              if(rq_write_lgn[index] == -1 and rq_read_lgn[index] != -1):
                  rq_write_lgn[index] = rq_read_lgn[index]
                  rq_write_lgn_previous[index] = rq_read_lgn[index]
              elif(rq_write_lgn_previous[index] == -1 and rq_read_lgn[index] != -1):
                  rq_write_lgn_previous[index] = rq_read_lgn[index]
              end

              if(rq_write_msc[index] == -1 and rq_read_msc[index] != -1):
                  rq_write_msc[index] = rq_read_msc[index]
                  rq_write_msc_previous[index] = rq_read_msc[index]
              elif(rq_write_msc_previous[index] == -1 and rq_read_msc[index] != -1):
                  rq_write_msc_previous[index] = rq_read_msc[index]
              end

              if(rq_write_mod[index] == -1 and rq_read_mod[index] != -1):
                  rq_write_mod[index] = rq_read_mod[index]
                  rq_write_mod_previous[index] = rq_read_mod[index]
              elif(rq_write_mod_previous[index] == -1 and rq_read_mod[index] != -1):
                  rq_write_mod_previous[index] = rq_read_mod[index]
              end

          end
          index = index + 1
      end
  end

  def rq_comm_set_var(var, value=0, gripper_socket="1"):
      socket_set_var(var, value, gripper_socket)
      return socket_read_byte_list(3, gripper_socket)
  end

  def rq_comm_set_pos_spe_for(pos=0, speed=0, force=0, gripper_socket="1"):
      socket_send_string("SET POS", gripper_socket)
      socket_send_byte(32, gripper_socket)
      socket_send_string(pos, gripper_socket)
      socket_send_byte(32, gripper_socket)
      socket_send_string("SPE", gripper_socket)
      socket_send_byte(32, gripper_socket)
      socket_send_string(speed, gripper_socket)
      socket_send_byte(32, gripper_socket)
      socket_send_string("FOR", gripper_socket)
      socket_send_byte(32, gripper_socket)
      socket_send_string(force, gripper_socket)
      socket_send_byte(10, gripper_socket)
      return socket_read_byte_list(3, gripper_socket)
  end

  def rq_comm_read_variables():
      index = 0

      while(index <= 3):
          socket = rq_index_to_socket(index)

          if(gripper_connected[index]):

              if(rq_read_act_req[index]):
                  rq_read_act[index] = socket_get_var("ACT", socket)
                  rq_read_act_req[index] = False
              end

              if(rq_read_gto_req[index]):
                  rq_read_gto[index] = socket_get_var("GTO", socket)
                  rq_read_gto_req[index] = False
              end

              if(rq_read_pre_req[index]):
                  rq_read_pre[index] = socket_get_var("PRE", socket)
                  rq_read_pre_req[index] = False
              end

              if(rq_read_pos_req[index]):
                  rq_read_pos[index] = socket_get_var("POS", socket)
                  rq_read_pos_req[index] = False
              end

              if(rq_read_spe_req[index]):
                  rq_read_spe[index] = socket_get_var("SPE", socket)
                  rq_read_spe_req[index] = False
              end

              if(rq_read_for_req[index]):
                  rq_read_for[index] = socket_get_var("FOR", socket)
                  rq_read_for_req[index] = False
              end

              if(rq_read_obj_req[index]):
                  rq_read_obj[index] = socket_get_var("OBJ", socket)
                  rq_read_obj_req[index] = False
              end

              if(rq_read_sta_req[index]):
                  rq_read_sta[index] = socket_get_var("STA", socket)
                  rq_read_sta_req[index] = False
              end

              if(rq_read_mod_req[index]):
                  rq_read_mod[index] = socket_get_var("MOD", socket)
                  rq_read_mod_req[index] = False
              end

              if(rq_read_flt_req[index]):
                  rq_read_flt[index] = socket_get_var("FLT",socket)
                  rq_read_flt_req[index] = False
              end

              if(rq_read_lbp_req[index]):
                  rq_read_lbp[index] = socket_get_var("LBP", socket)
                  rq_read_lbp_req[index] = False
              end

              if(rq_read_lrd_req[index]):
                  rq_read_lrd[index] = socket_get_var("LRD", socket)
                  rq_read_lrd_req[index] = False
              end

              if(rq_read_lbl_req[index]):
                  rq_read_lbl[index] = socket_get_var("LBL",socket)
                  rq_read_lbl_req[index] = False
              end

              if(rq_read_lgn_req[index]):
                  rq_read_lgn[index] = socket_get_var("LGN", socket)
                  rq_read_lgn_req[index] = False
              end

              if(rq_read_msc_req[index]):
                  rq_read_msc[index] = socket_get_var("MSC", socket)
                  rq_read_msc_req[index] = False
              end

              if(rq_read_cou_req[index]):
                  rq_read_cou[index] = socket_get_var("COU", socket)
                  rq_read_cou_req[index] = False
              end

              if(rq_read_ncy_req[index]):
                  rq_read_ncy[index] = socket_get_var("NCY", socket)
                  rq_read_ncy_req[index] = False
              end

              if(rq_read_dst_req[index]):
                  rq_read_dst[index] = socket_get_var("DST", socket)
                  rq_read_dst_req[index] = False
              end

              if(rq_read_pco_req[index]):
                  rq_read_pco[index] = socket_get_var("PCO", socket)
                  rq_read_pco_req[index] = False
              end
          end
          index = index + 1
      end
  end

  def rq_comm_read_constants():

      if(gripper_connected[0]):
          while(rq_read_snu_1 == rq_string_initial_value):
              socket_send_string("GET SNU", "1")
              rq_read_snu_1 = socket_read_string("1")
          end

          while(rq_read_fwv_1 == rq_string_initial_value):
              socket_send_string("GET FWV", "1")
              rq_read_fwv_1 = socket_read_string("1")
          end

          while(rq_read_ver_1 == rq_string_initial_value):
              socket_send_string("GET VER", "1")
              rq_read_ver_1 = socket_read_string("1")
          end
      end

      if(gripper_connected[1]):
          while(rq_read_snu_2 == rq_string_initial_value):
              socket_send_string("GET SNU", "2")
              rq_read_snu_2 = socket_read_string("2")
          end

          while(rq_read_fwv_2 == rq_string_initial_value):
              socket_send_string("GET FWV", "2")
              rq_read_fwv_2 = socket_read_string("2")
          end

          while(rq_read_ver_2 == rq_string_initial_value):
              socket_send_string("GET VER", "2")
              rq_read_ver_2 = socket_read_string("2")
          end
      end

      if(gripper_connected[2]):
          while(rq_read_snu_3 == rq_string_initial_value):
              socket_send_string("GET SNU", "3")
              rq_read_snu_3 = socket_read_string("3")
          end

          while(rq_read_fwv_3 == rq_string_initial_value):
              socket_send_string("GET FWV", "3")
              rq_read_fwv_3 = socket_read_string("3")
          end

          while(rq_read_ver_3 == rq_string_initial_value):
              socket_send_string("GET VER", "3")
              rq_read_ver_3 = socket_read_string("3")
          end
      end

      if(gripper_connected[3]):
          while(rq_read_snu_4 == rq_string_initial_value):
              socket_send_string("GET SNU", "4")
              rq_read_snu_4 = socket_read_string("4")
          end

          while(rq_read_fwv_4 == rq_string_initial_value):
              socket_send_string("GET FWV", "4")
              rq_read_fwv_4 = socket_read_string("4")
          end

          while(rq_read_ver_4 == rq_string_initial_value):
              socket_send_string("GET VER", "4")
              rq_read_ver_4 = socket_read_string("4")
          end
      end
  end

  def rq_comm_write_variables():
      index = 0

      while(index <= 3):
          socket = rq_index_to_socket(index)

          if(gripper_connected[index]):

              if(rq_write_act_request[index]):
                  if(is_ack(rq_comm_set_var("ACT", rq_write_act[index], socket))):
                      rq_write_act_previous[index] = rq_write_act[index]
                      rq_write_act_request[index] = False
                  end
              end

              if(rq_write_gto_request[index]):
                  if(is_ack(rq_comm_set_var("GTO", rq_write_gto[index], socket))):
                      rq_write_gto_previous[index] = rq_write_gto[index]
                      rq_write_gto_request[index] = False
                  end
              end

              if(rq_write_atr_request[index]):
                  if(is_ack(rq_comm_set_var("ATR", rq_write_atr[index], socket))):
                      rq_write_atr_previous[index] = rq_write_atr[index]
                      rq_write_atr_request[index] = False
                  end
              end

              if(rq_write_ard_request[index]):
                  if(is_ack(rq_comm_set_var("ARD", rq_write_ard[index], socket))):
                      rq_write_ard_previous[index] = rq_write_ard[index]
                      rq_write_ard_request[index] = False
                  end
              end

              if(rq_write_pos_request[index]):
                  if(is_ack(rq_comm_set_pos_spe_for(rq_write_pos[index], rq_write_spe[index], rq_write_for[index], socket))):
                      rq_write_pos_previous[index] = rq_write_pos[index]
                      rq_write_spe_previous[index] = rq_write_spe[index]
                      rq_write_for_previous[index] = rq_write_for[index]
                      rq_write_pos_request[index] = False
                  end
              end

              if(rq_write_lbp_request[index]):
                  if(is_ack(rq_comm_set_var("LBP", rq_write_lbp[index], socket))):
                      rq_write_lbp_previous[index] = rq_write_lbp[index]
                      rq_write_lbp_request[index] = False
                  end
              end

              if(rq_write_lrd_request[index]):
                  if(is_ack(rq_comm_set_var("LRD", rq_write_lrd[index], socket))):
                      rq_write_lrd_previous[index] = rq_write_lrd[index]
                      rq_write_lrd_request[index] = False
                  end
              end

              if(rq_write_lbl_request[index]):
                  if(is_ack(rq_comm_set_var("LBL", rq_write_lbl[index], socket))):
                      rq_write_lbl_previous[index] = rq_write_lbl[index]
                      rq_write_lbl_request[index] = False
                  end
              end

              if(rq_write_lgn_request[index]):
                  if(is_ack(rq_comm_set_var("LGN", rq_write_lgn[index], socket))):
                      rq_write_lgn_previous[index] = rq_write_lgn[index]
                      rq_write_lgn_request[index] = False
                  end
              end

              if(rq_write_msc_request[index]):
                  if(is_ack(rq_comm_set_var("MSC", rq_write_msc[index], socket))):
                      rq_write_msc_previous[index] = rq_write_msc[index]
                      rq_write_msc_request[index] = False
                  end
              end

              if(rq_write_mod_request[index]):
                  if(is_ack(rq_comm_set_var("MOD", rq_write_mod[index], socket))):
                      rq_write_mod_previous[index] = rq_write_mod[index]
                      rq_write_mod_request[index] = False
                  end
              end
          end
          index = index + 1
      end
  end

  def rq_activate(gripper_socket="1"):
      if (not rq_is_gripper_activated(gripper_socket)):
          rq_reset(gripper_socket)

          while(not rq_get_var("ACT", 1, gripper_socket) == 0 or not rq_get_var("STA", 1, gripper_socket) == 0):
              rq_reset(gripper_socket)
              sync()
          end

          rq_set_var("ACT",1, gripper_socket)
      end
  end

  def rq_activate_and_wait(gripper_socket="1"):
      if (not rq_is_gripper_activated(gripper_socket)):
          rq_activate(gripper_socket)
          sleep(1.0)

          while(not rq_get_var("ACT", 1, gripper_socket) == 1 or not rq_get_var("STA", 1, gripper_socket) == 3):
              sleep(0.1)
          end

          sleep(0.5)
      end
  end

  def rq_activate_all_grippers(reset=False):
      if(gripper_connected[0]):
          rq_reset_and_activate("1", reset)
      end

      if(gripper_connected[1]):
          rq_reset_and_activate("2", reset)
      end

      if(gripper_connected[2]):
          rq_reset_and_activate("3", reset)
      end

      if(gripper_connected[3]):
          rq_reset_and_activate("4", reset)
      end
  end

  def rq_reset_and_activate(gripper_socket="1", reset=False):
      if(reset):
          rq_reset(gripper_socket)
          rq_activate_and_wait(gripper_socket)
      elif(not rq_is_gripper_activated(gripper_socket)):
          rq_activate_and_wait(gripper_socket)
      end
  end

  def rq_reset(gripper_socket="1"):
      rq_set_var("ACT", 0, gripper_socket)
      rq_set_var("ATR", 0, gripper_socket)

      while(not rq_get_var("ACT", 1, gripper_socket) == 0 or not rq_get_var("STA", 1, gripper_socket) == 0):
          rq_set_var("ACT", 0, gripper_socket)
          rq_set_var("ATR", 0, gripper_socket)
          sync()
      end

      sleep(0.5)
  end

  def rq_auto_release_open_and_wait(gripper_socket="1"):
      rq_set_var("ATR",0, gripper_socket)
      rq_set_var("ARD",0, gripper_socket)
      rq_set_var("ACT",1, gripper_socket)
      sleep(0.1)
      rq_set_var("ATR",1, gripper_socket)

      rq_wait_autorelease_completed(gripper_socket)
  end

  def rq_auto_release_close_and_wait(gripper_socket="1"):
      rq_set_var("ATR",0, gripper_socket)
      rq_set_var("ARD",1, gripper_socket)
      rq_set_var("ACT",1, gripper_socket)
      sleep(0.1)
      rq_set_var("ATR",1, gripper_socket)

      rq_wait_autorelease_completed(gripper_socket)
  end

  def rq_wait_autorelease_completed(gripper_socket="1"):
      remainingRetries = 20
      gFLT = rq_get_var("FLT", 2, gripper_socket)

      while(not is_FLT_autorelease_in_progress(gFLT) and remainingRetries > 0):
          remainingRetries = remainingRetries - 1
          gFLT = rq_get_var("FLT", 2, gripper_socket)
          sleep(0.1)
      end

      remainingRetries = 100
      gFLT = rq_get_var("FLT", 2, gripper_socket)

      while(not is_FLT_autorelease_completed(gFLT) and remainingRetries > 0):
          remainingRetries = remainingRetries - 1
          gFLT = rq_get_var("FLT", 2, gripper_socket)
          sleep(0.1)
      end
  end

  def rq_set_force(force, gripper_socket="1"):
      force = floor(scale(force, [0, 255], [0.0, 255.0]))
      rq_set_var("FOR", force, gripper_socket)
  end

  def rq_set_speed(speed, gripper_socket="1"):
      speed = floor(scale(speed, [0, 255], [0.0, 255.0]))
      rq_set_var("SPE", speed, gripper_socket)
  end

  def rq_open(gripper_socket="1"):
      rq_move(0, gripper_socket)
  end

  def rq_close(gripper_socket="1"):
      rq_move(255, gripper_socket)
  end

  def rq_open_and_wait(gripper_socket="1"):
      rq_move_and_wait(0, gripper_socket)
  end

  def rq_close_and_wait(gripper_socket="1"):
      rq_move_and_wait(255, gripper_socket)
  end

  def rq_move(pos, gripper_socket="1"):
      rq_set_pos(pos, gripper_socket)
      rq_go_to(gripper_socket)
  end

  def rq_move_and_wait(pos, gripper_socket="1"):
      rq_move(pos, gripper_socket)

      while (not rq_is_motion_complete(gripper_socket)):
          # wait for motion completed
          sync()
      end
  end

  def rq_wait_for_pos_request(pos, gripper_socket="1"):
      gPRE = rq_get_var("PRE", 3, gripper_socket)

      while (gPRE != pos):
          rq_set_var("POS", pos, gripper_socket)
          sync()
          gPRE = rq_get_var("PRE", 3, gripper_socket)
      end
  end

  def rq_wait_pos_spe_for_request(pos, speed, force, gripper_socket="1"):
      gPRE = rq_get_var("PRE", 3, gripper_socket)

      while (gPRE != pos):
          rq_set_pos_spe_for_var(pos, speed, force, gripper_socket)
          sync()
          gPRE = rq_get_var("PRE", 3, gripper_socket)
      end
  end

  def rq_wait_for_pos(pos, gripper_socket="1"):
      rq_wait_for_pos_request(pos, gripper_socket)

      # Wait for the gripper motion to complete
      while (not rq_is_motion_complete(gripper_socket)):
          # wait for motion completed
          sync()
          rq_set_var("GTO", 1, gripper_socket)
      end
  end

  def rq_wait(gripper_socket="1"):
      # Wait for the gripper motion to complete
      while (not rq_is_motion_complete(gripper_socket)):
          sync()
          # The following patch is for Robotiq's Camera issue when communication is lost, but not the activation
          # the communication driver reset the GTO bit
          rq_set_var("GTO", 1, gripper_socket)
      end
  end

  def rq_wait_for_object_detected(gripper_socket="1"):
      # Wait the object detection
      while (not rq_is_object_detected(gripper_socket)):
          sync()
      end
  end

  # set the position
  def rq_set_pos(pos, gripper_socket="1"):
      pos = floor(scale(pos, [0, 255], [0.0, 255.0]))
      rq_set_var("POS", pos, gripper_socket)
      rq_wait_for_pos_request(pos, gripper_socket)
  end

  def rq_set_pos_spd_for(pos, speed, force, gripper_socket="1"):
      pos = floor(scale(pos, [0, 255], [0.0, 255.0]))
      speed = floor(scale(speed, [0, 255], [0.0, 255.0]))
      force = floor(scale(force, [0, 255], [0.0, 255.0]))

      rq_set_pos_spe_for_var(pos, speed, force, gripper_socket)
  end

  def rq_set_gripper_max_current_mA(current_mA, gripper_socket="1"):
      current = floor(current_mA / 10)

      rq_set_var("MSC", current, gripper_socket)
      current_read = rq_get_var("MSC", 1, gripper_socket)

      while(current_read != current):
          rq_set_var("MSC", current, gripper_socket)
          current_read = rq_get_var("MSC", 1, gripper_socket)
      end
  end

  def rq_set_gripper_mode(mode, gripper_socket="1"):
      rq_set_var("MOD", mode, gripper_socket)
  end

  def rq_set_gripper_max_cur(current_mA, gripper_socket="1"):
      rq_set_gripper_max_current_mA(current_mA, gripper_socket)
  end

  def rq_get_gripper_max_current_mA(gripper_socket="1"):
      current = rq_get_var("MSC", 1, gripper_socket)

      if(current == -1):
          current_mA = current
      else:
          current_mA = current * 10
      end

      return current_mA
  end

  def rq_get_gripper_max_cur(gripper_socket="1"):
      return rq_get_gripper_max_current_mA(gripper_socket)
  end

  def rq_set_max_current_for_all_grippers():
      current_mA = rq_get_max_current_mA()

      if(gripper_connected[0]):
          rq_set_gripper_max_current_mA(current_mA, "1")
      end

      if(gripper_connected[1]):
          rq_set_gripper_max_current_mA(current_mA, "2")
      end

      if(gripper_connected[2]):
          rq_set_gripper_max_current_mA(current_mA, "3")
      end

      if(gripper_connected[3]):
          rq_set_gripper_max_current_mA(current_mA, "4")
      end
  end

  def rq_get_max_current_mA():
      max_current_mA = 0

      if(rq_current_limit_enabled):
          nb_connected_grippers = rq_get_nb_connected_grippers()

          if(nb_connected_grippers == 1):
              max_current_mA = 600
          elif(nb_connected_grippers > 1):
              max_current_mA = 450
          end
      else:

      end

      return max_current_mA
  end

  def rq_get_nb_connected_grippers():
      nb_connected_grippers = 0

      if(gripper_connected[0]):
          nb_connected_grippers = nb_connected_grippers + 1
      end

      if(gripper_connected[1]):
          nb_connected_grippers = nb_connected_grippers + 1
      end

      if(gripper_connected[2]):
          nb_connected_grippers = nb_connected_grippers + 1
      end

      if(gripper_connected[3]):
          nb_connected_grippers = nb_connected_grippers + 1
      end

      return nb_connected_grippers
  end

  def rq_list_of_bytes_to_value(list_of_bytes):
      value = -1

      # response list length
      if (list_of_bytes[0] == 1):
          value = list_of_bytes[1] - 48
      elif (list_of_bytes[0] == 2):
          value = (list_of_bytes[1] - 48) * 10 + (list_of_bytes[2] - 48)
      elif (list_of_bytes[0] == 3):
          value = (list_of_bytes[1] - 48) * 100 + (list_of_bytes[2] - 48) * 10 + (list_of_bytes[3] - 48)
      end

      return value
  end

  def rq_is_motion_complete(gripper_socket="1"):
      gOBJ = rq_get_var("OBJ", 1, gripper_socket)
      sync()
      return is_OBJ_gripper_at_position(gOBJ) or is_OBJ_object_detected(gOBJ)
  end

  def rq_is_gripper_activated(gripper_socket="1"):
      gSTA = rq_get_var("STA", 1, gripper_socket)
      sync()
      return is_STA_gripper_activated(gSTA)
  end

  def rq_is_object_detected(gripper_socket="1"):
      gOBJ = rq_get_var("OBJ", 1, gripper_socket)
      sync()
      return is_OBJ_object_detected(gOBJ)
  end

  def rq_current_pos(gripper_socket="1"):
      gPOS = rq_get_var("POS", 1, gripper_socket)
      sync()
      return gPOS
  end

  def rq_motor_current(gripper_socket="1"):
      rq_current = rq_get_var("COU", 1, gripper_socket)
      sync()
      return rq_current * 10
  end

  def rq_print_connected_grippers():
      if(gripper_connected[0]):
          textmsg("Gripper 1 : ", "connected and socket open.")
      end

      if (gripper_connected[1]):
          textmsg("Gripper 2 : ", "connected and socket open.")
      end

      if (gripper_connected[2]):
          textmsg("Gripper 3 : ", "connected and socket open.")
      end

      if (gripper_connected[3]):
          textmsg("Gripper 4 : ", "connected and socket open.")
      end
  end

  def rq_print_gripper_fault_code(gripper_socket="1"):
      gFLT = rq_get_var("FLT", 2, gripper_socket)

      if(is_FLT_no_fault(gFLT)):
          textmsg("Gripper Fault : ", "No Fault (0x00)")
      elif (is_FLT_action_delayed(gFLT)):
          textmsg("Gripper Fault : ", "Priority Fault: Action delayed, initialization must be completed prior to action (0x05)")
      elif (is_FLT_not_activated(gFLT)):
          textmsg("Gripper Fault : ", "Priority Fault: The activation must be set prior to action (0x07)")
      elif (is_FLT_autorelease_in_progress(gFLT)):
          textmsg("Gripper Fault : ", "Minor Fault: Automatic release in progress (0x0B)")
      elif (is_FLT_overcurrent(gFLT)):
          textmsg("Gripper Fault : ", "Minor Fault: Overcurrent protection triggered (0x0E)")
      elif (is_FLT_autorelease_completed(gFLT)):
          textmsg("Gripper Fault : ", "Major Fault: Automatic release completed (0x0F)")
      else:
          textmsg("Gripper Fault : ", "Unknown Fault")
      end
  end

  def rq_print_gripper_num_cycles(gripper_socket="1"):
      num_cycles = rq_get_var("NCY", 1, gripper_socket)

      if(num_cycles == -1):
          textmsg("Gripper Cycle Number : ", "Number of cycles is unreachable.")
      else:
          textmsg("Gripper Cycle Number : ", num_cycles)
      end
  end

  def rq_print_gripper_driver_state(gripper_socket="1"):
      driver_state = rq_get_var("DST", 1, gripper_socket)

      if(driver_state == 0):
          textmsg("Gripper Driver State : ", "RQ_STATE_INIT")
      elif(driver_state == 1):
          textmsg("Gripper Driver State : ", "RQ_STATE_LISTEN")
      elif(driver_state == 2):
          textmsg("Gripper Driver State : ", "RQ_STATE_READ_INFO")
      elif(driver_state == 3):
          textmsg("Gripper Driver State : ", "RQ_STATE_ACTIVATION")
      else:
          textmsg("Gripper Driver State : ", "RQ_STATE_RUN")
      end
  end

  def rq_print_gripper_serial_number(gripper_socket="1"):
      serial_number = rq_get_var_string("SNU", 1, gripper_socket)
      textmsg("Gripper Serial Number : ", serial_number)
  end

  def rq_print_gripper_firmware_version(gripper_socket="1"):
      firmware_version = rq_get_var_string("FWV", 1, gripper_socket)
      textmsg("Gripper Firmware Version : ", firmware_version)
  end

  def rq_print_gripper_driver_version(gripper_socket="1"):
      driver_version = rq_get_var_string("VER", 1, gripper_socket)
      textmsg("Gripper Driver Version : ", driver_version)
  end

  def rq_print_gripper_connection_state(gripper_socket="1"):
      connection_state = rq_get_var("PCO", 1, gripper_socket)

      if (connection_state == 0):
          textmsg("Gripper Connection State : ", "No connection problem detected")
      else:
          textmsg("Gripper Connection State : ", "Connection problem detected")
      end
  end

  # Returns True if list_of_bytes is [3, 'a', 'c', 'k']
  def is_ack(list_of_bytes):

      # list length is not 3
      if (list_of_bytes[0] != 3):
          return False
      end

      # first byte not is 'a'?
      if (list_of_bytes[1] != 97):
          return False
      end

      # first byte not is 'c'?
      if (list_of_bytes[2] != 99):
          return False
      end

      # first byte not is 'k'?
      if (list_of_bytes[3] != 107):
          return False
      end

      return True
  end

  # Returns True if list_of_bytes is not [3, 'a', 'c', 'k']
  def is_not_ack(list_of_bytes):
      if (is_ack(list_of_bytes)):
          return False
      else:
          return True
      end
  end

  def is_STA_gripper_activated (gSTA):
      if (gSTA == 3):
          return True
      end

      return False
  end

  def is_OBJ_object_detected (gOBJ):
      if (gOBJ == 1 or gOBJ == 2):
          return True
      end

      return False
  end

  def is_OBJ_gripper_at_position (gOBJ):
      if (gOBJ == 3):
          return True
      end

      return False
  end

  def is_not_OBJ_gripper_at_position (gOBJ):
      if (is_OBJ_gripper_at_position(gOBJ)):
          return False
      else:
          return True
      end
  end

  #### GTO Section ####
  def rq_stop(gripper_socket="1"):
      rq_set_var("GTO", 0, gripper_socket)
  end

  def rq_set_GTO_and_wait(value, gripper_socket="1"):
      rq_set_var("GTO" ,value, gripper_socket)
      while(not is_GTO(value, rq_get_var("GTO", 1, gripper_socket))):
        sync()
      end
  end

  def rq_go_to(gripper_socket="1"):
      rq_set_var("GTO", 1, gripper_socket)
  end


  def is_GTO(goto_value, rGTO):
      return rGTO == goto_value
  end
  #### GTO Section ####

  def is_FLT_no_fault(gFLT):
      return gFLT == 0
  end

  def is_FLT_warning(gFLT):
      return gFLT >= 1 and gFLT <= 7
  end

  def is_FLT_faulted(gFLT):
      return gFLT >= 8
  end

  def is_FLT_action_delayed(gFLT):
      return gFLT == 5
  end

  def is_FLT_not_activated(gFLT):
      return gFLT == 7
  end

  def is_FLT_autorelease_in_progress(gFLT):
      return gFLT == 11
  end

  def is_FLT_overcurrent(gFLT):
      return gFLT == 14
  end

  def is_FLT_autorelease_completed(gFLT):
      return gFLT == 15
  end

  def rq_set_var(var_name, var_value, gripper_socket="1"):
      index = rq_socket_to_index(gripper_socket)

      enter_critical

      if (var_name == "ACT"):
          rq_write_act[index] = var_value
          rq_write_act_request[index] = True
      elif (var_name == "GTO"):
          rq_write_gto[index] = var_value
          rq_write_gto_request[index] = True
      elif (var_name == "ATR"):
          rq_write_atr[index] = var_value
          rq_write_atr_request[index] = True
      elif (var_name == "ARD"):
          rq_write_ard[index] = var_value
          rq_write_ard_request[index] = True
      elif (var_name == "FOR"):
          rq_write_for[index] = var_value
          rq_write_pos_request[index] = True
      elif (var_name == "SPE"):
          rq_write_spe[index] = var_value
          rq_write_pos_request[index] = True
      elif (var_name == "POS"):
          rq_write_pos[index] = var_value
          rq_write_pos_request[index] = True
      elif (var_name == "LBP"):
          rq_write_lbp[index] = var_value
          rq_write_lbp_request[index] = True
      elif (var_name == "LRD"):
          rq_write_lrd[index] = var_value
          rq_write_lrd_request[index] = True
      elif (var_name == "LBL"):
          rq_write_lbl[index] = var_value
          rq_write_lbl_request[index] = True
      elif (var_name == "LGN"):
          rq_write_lgn[index] = var_value
          rq_write_lgn_request[index] = True
      elif (var_name == "MSC"):
          rq_write_msc[index] = var_value
          rq_write_msc_request[index] = True
      elif (var_name == "MOD"):
          rq_write_mod[index] = var_value
          rq_write_mod_request[index] = True
      end

      exit_critical

      if (var_name == "ACT"):
          while(rq_write_act_request[index]):
              sync()
          end
      elif (var_name == "GTO"):
          while(rq_write_gto_request[index]):
              sync()
          end
      elif (var_name == "ATR"):
          while(rq_write_atr_request[index]):
              sync()
          end
      elif (var_name == "ARD"):
          while(rq_write_ard_request[index]):
              sync()
          end
      elif (var_name == "FOR"):
          while(rq_write_pos_request[index]):
              sync()
          end
      elif (var_name == "SPE"):
          while(rq_write_pos_request[index]):
              sync()
          end
      elif (var_name == "POS"):
          while(rq_write_pos_request[index]):
              sync()
          end
      elif (var_name == "LBP"):
          while(rq_write_lbp_request[index]):
              sync()
          end
      elif (var_name == "LRD"):
          while(rq_write_lrd_request[index]):
              sync()
          end
      elif (var_name == "LBL"):
          while(rq_write_lbl_request[index]):
              sync()
          end
      elif (var_name == "LGN"):
          while(rq_write_lgn_request[index]):
              sync()
          end
      elif (var_name == "MSC"):
          while(rq_write_msc_request[index]):
              sync()
          end
      elif (var_name == "MOD"):
          while(rq_write_mod_request[index]):
              sync()
          end
      end
  end

  def rq_set_pos_spe_for_var(pos, speed, force, gripper_socket="1"):
      index = rq_socket_to_index(gripper_socket)

      enter_critical

      rq_write_for[index] = force
      rq_write_spe[index] = speed
      rq_write_pos[index] = pos
      rq_write_pos_request[index] = True

      exit_critical
  end

  def rq_get_var(var_name, nbr_bytes, gripper_socket="1"):
      index = rq_socket_to_index(gripper_socket)
      var_value = -1

      if (var_name == "ACT"):
          enter_critical
          rq_read_act_req[index] = True
          exit_critical
          while(rq_read_act_req[index]):
              sync()
          end
          var_value = rq_read_act[index]

      elif (var_name == "GTO"):
          enter_critical
          rq_read_gto_req[index] = True
          exit_critical
          while(rq_read_gto_req[index]):
              sync()
          end
          var_value = rq_read_gto[index]

      elif (var_name == "FOR"):
          enter_critical
          rq_read_for_req[index] = True
          exit_critical
          while(rq_read_for_req[index]):
              sync()
          end
          var_value = rq_read_for[index]

      elif (var_name == "SPE"):
          enter_critical
          rq_read_spe_req[index] = True
          exit_critical
          while(rq_read_spe_req[index]):
              sync()
          end
          var_value = rq_read_spe[index]

      elif (var_name == "OBJ"):
          enter_critical
          rq_read_obj_req[index] = True
          exit_critical
          while(rq_read_obj_req[index]):
              sync()
          end
          var_value = rq_read_obj[index]

      elif (var_name == "STA"):
          enter_critical
          rq_read_sta_req[index] = True
          exit_critical
          while(rq_read_sta_req[index]):
              sync()
          end
          var_value = rq_read_sta[index]

      elif (var_name == "FLT"):
          enter_critical
          rq_read_flt_req[index] = True
          exit_critical
          while(rq_read_flt_req[index]):
              sync()
          end
          var_value = rq_read_flt[index]

      elif (var_name == "POS"):
          enter_critical
          rq_read_pos_req[index] = True
          exit_critical
          while(rq_read_pos_req[index]):
              sync()
          end
          var_value = rq_read_pos[index]

      elif (var_name == "PRE"):
          enter_critical
          rq_read_pre_req[index] = True
          exit_critical
          while(rq_read_pre_req[index]):
              sync()
          end
          var_value = rq_read_pre[index]

      elif (var_name == "LBP"):
          enter_critical
          rq_read_lbp_req[index] = True
          exit_critical
          while(rq_read_lbp_req[index]):
              sync()
          end
          var_value = rq_read_lbp[index]

      elif (var_name == "LRD"):
          enter_critical
          rq_read_lrd_req[index] = True
          exit_critical
          while(rq_read_lrd_req[index]):
              sync()
          end
          var_value = rq_read_lrd[index]

      elif (var_name == "LBL"):
          enter_critical
          rq_read_lbl_req[index] = True
          exit_critical
          while(rq_read_lbl_req[index]):
              sync()
          end
          var_value = rq_read_lbl[index]

      elif (var_name == "LGN"):
          enter_critical
          rq_read_lgn_req[index] = True
          exit_critical
          while(rq_read_lgn_req[index]):
              sync()
          end
          var_value = rq_read_lgn[index]

      elif (var_name == "MSC"):
          enter_critical
          rq_read_msc_req[index] = True
          exit_critical
          while(rq_read_msc_req[index]):
              sync()
          end
          var_value = rq_read_msc[index]

      elif (var_name == "MOD"):
          enter_critical
          rq_read_mod_req[index] = True
          exit_critical
          while(rq_read_mod_req[index]):
              sync()
          end
          var_value = rq_read_mod[index]

      elif (var_name == "NCY"):
          enter_critical
          rq_read_ncy_req[index] = True
          exit_critical
          while(rq_read_ncy_req[index]):
              sync()
          end
          var_value = rq_read_ncy[index]

      elif (var_name == "PCO"):
          enter_critical
          rq_read_pco_req[index] = True
          exit_critical
          while(rq_read_pco_req[index]):
              sync()
          end
          var_value = rq_read_pco[index]

      elif (var_name == "DST"):
          enter_critical
          rq_read_dst_req[index] = True
          exit_critical
          while(rq_read_dst_req[index]):
              sync()
          end
          var_value = rq_read_dst[index]

      end

      return var_value
  end

  def rq_get_var_string(var_name, nbr_bytes, gripper_socket="1"):
      index = rq_socket_to_index(gripper_socket)
      var_value = ""

      enter_critical

      if (var_name == "SNU"):
          if(gripper_socket == "1"):
              var_value = rq_read_snu_1
          elif(gripper_socket == "2"):
              var_value = rq_read_snu_2
          elif(gripper_socket == "3"):
              var_value = rq_read_snu_3
          elif(gripper_socket == "4"):
              var_value = rq_read_snu_4
          end
      elif (var_name == "FWV"):
          if(gripper_socket == "1"):
              var_value = rq_read_fwv_1
          elif(gripper_socket == "2"):
              var_value = rq_read_fwv_2
          elif(gripper_socket == "3"):
              var_value = rq_read_fwv_3
          elif(gripper_socket == "4"):
              var_value = rq_read_fwv_4
          end
      elif (var_name == "VER"):
          if(gripper_socket == "1"):
              var_value = rq_read_ver_1
          elif(gripper_socket == "2"):
              var_value = rq_read_ver_2
          elif(gripper_socket == "3"):
              var_value = rq_read_ver_3
          elif(gripper_socket == "4"):
              var_value = rq_read_ver_4
          end
      end

      exit_critical

      return var_value
  end

  def rq_is_object_validated(gripper_selected, gripper_socket="1"):
      if(gripper_selected):
          if(rq_is_object_detected(gripper_socket)):
              return True
          else:
              return False
          end
      else:
          return True
      end
  end

  ############################################
  # normalized functions (maps 0-100 to 0-255)
  ############################################
  def rq_set_force_norm(force_norm, gripper_socket="1"):
      force_gripper = norm_to_gripper(force_norm)
      rq_set_force(force_gripper, gripper_socket)
  end

  def rq_set_speed_norm(speed_norm, gripper_socket="1"):
      speed_gripper = norm_to_gripper(speed_norm)
      rq_set_speed(speed_gripper, gripper_socket)
  end

  def rq_move_norm(pos_norm, gripper_socket="1"):
      pos_gripper = norm_to_gripper(pos_norm)
      rq_move(pos_gripper, gripper_socket)
  end

  def rq_move_and_wait_norm(pos_norm, gripper_socket="1"):
      pos_gripper = norm_to_gripper(pos_norm)
      rq_move_and_wait(pos_gripper, gripper_socket)
  end

  def rq_set_pos_norm(pos_norm, gripper_socket="1"):
      pos_gripper = norm_to_gripper(pos_norm)
      rq_set_pos(pos_gripper, gripper_socket)
  end

  def rq_current_pos_norm(gripper_socket="1"):
      pos_gripper = rq_current_pos(gripper_socket)
      pos_norm = gripper_to_norm(pos_gripper)
      return pos_norm
  end

  def gripper_to_norm(value_gripper):
      value_norm = (value_gripper / 255) * 100
      return floor(value_norm)
  end

  def norm_to_gripper(value_norm):
      value_gripper = (value_norm / 100) * 255
      return ceil(value_gripper)
  end

  def rq_get_position():
      return rq_current_pos_norm()
  end

  def rq_gripper_led_on(gripper_socket="1"):
      rq_set_var("LBP",0, gripper_socket)
  end

  def rq_gripper_led_off(gripper_socket="1"):
      rq_set_var("LBP",1, gripper_socket)
      rq_set_var("LRD",0, gripper_socket)
      rq_set_var("LBL",0, gripper_socket)
      rq_set_var("LGN",0, gripper_socket)
  end

  def rq_gripper_led_force_red(gripper_socket="1"):
      rq_set_var("LBP",1, gripper_socket)
      rq_set_var("LRD",1, gripper_socket)
      rq_set_var("LBL",0, gripper_socket)
      rq_set_var("LGN",0, gripper_socket)
  end

  def rq_gripper_led_force_blue(gripper_socket="1"):
      rq_set_var("LBP",1, gripper_socket)
      rq_set_var("LRD",0, gripper_socket)
      rq_set_var("LBL",1, gripper_socket)
      rq_set_var("LGN",0, gripper_socket)
  end

  def rq_gripper_led_force_green(gripper_socket="1"):
      rq_set_var("LBP",1, gripper_socket)
      rq_set_var("LRD",0, gripper_socket)
      rq_set_var("LBL",0, gripper_socket)
      rq_set_var("LGN",1, gripper_socket)
  end

  def rq_gripper_led_force_purple(gripper_socket="1"):
      rq_set_var("LBP",1, gripper_socket)
      rq_set_var("LRD",1, gripper_socket)
      rq_set_var("LBL",1, gripper_socket)
      rq_set_var("LGN",0, gripper_socket)
  end

  ############################################
  # mm/inches functions
  ############################################
  gripper_closed_norm = [100, 100, 100, 100]
  gripper_open_norm = [0, 0, 0, 0]
  gripper_closed_mm = [0, 0, 0, 0]
  gripper_open_mm = [50, 50, 50, 50]

  def rq_current_pos_mm(gripper_socket=1):
      pos_gripper = rq_current_pos(gripper_socket)
      pos_mm = gripper_to_mm(pos_gripper, gripper_socket)
      return round_value_2_dec(pos_mm)
  end

  def rq_current_pos_inches(gripper_socket=1):
      pos_gripper = rq_current_pos(gripper_socket)
      pos_mm = gripper_to_mm(pos_gripper, gripper_socket)
      pos_in = pos_mm / 25.4
      return round_value_2_dec(pos_in)
  end

  def rq_move_mm(pos_mm, gripper_socket=1):
      pos_gripper = mm_to_gripper(pos_mm, gripper_socket)
      rq_move(pos_gripper, gripper_socket)
  end

  def rq_move_and_wait_mm(pos_mm, gripper_socket=1):
      pos_gripper = mm_to_gripper(pos_mm, gripper_socket)
      rq_move_and_wait(pos_gripper, gripper_socket)
  end

  def rq_move_inches(pos_in, gripper_socket=1):
      pos_mm = pos_in * 25.4
      rq_move_mm(pos_mm, gripper_socket)
  end

  def rq_move_and_wait_inches(pos_in, gripper_socket=1):
      pos_mm = pos_in * 25.4
      rq_move_and_wait_mm(pos_mm, gripper_socket)
  end

  def get_closed_norm(gripper_socket):
      return gripper_closed_norm[gripper_socket - 1]
  end

  def get_open_norm(gripper_socket):
      return gripper_open_norm[gripper_socket - 1]
  end

  def get_closed_mm(gripper_socket):
      return gripper_closed_mm[gripper_socket - 1]
  end

  def get_open_mm(gripper_socket):
      return gripper_open_mm[gripper_socket - 1]
  end

  def set_closed_norm(closed_norm, gripper_socket):
      gripper_closed_norm[gripper_socket - 1] = closed_norm
  end

  def set_open_norm(open_norm, gripper_socket):
      gripper_open_norm[gripper_socket - 1] = open_norm
  end

  def set_closed_mm(closed_mm, gripper_socket):
      gripper_closed_mm[gripper_socket - 1] = closed_mm
  end

  def set_open_mm(open_mm, gripper_socket):
      gripper_open_mm[gripper_socket - 1] = open_mm
  end

  def gripper_to_mm(value_gripper, gripper_socket):
      closed_norm = get_closed_norm(gripper_socket)
      open_norm = get_open_norm(gripper_socket)
      closed_mm = get_closed_mm(gripper_socket)
      open_mm = get_open_mm(gripper_socket)

      value_norm = (value_gripper / 255) * 100

      slope = (closed_mm - open_mm) / (closed_norm - open_norm)
      value_mm = slope * (value_norm - closed_norm) + closed_mm

      if (value_mm > open_mm):
          value_mm_limited = open_mm
      elif (value_mm < closed_mm):
          value_mm_limited = closed_mm
      else:
          value_mm_limited = value_mm
      end

      return value_mm_limited
  end

  def mm_to_gripper(value_mm, gripper_socket):
      closed_norm = get_closed_norm(gripper_socket)
      open_norm = get_open_norm(gripper_socket)
      closed_mm = get_closed_mm(gripper_socket)
      open_mm = get_open_mm(gripper_socket)

      slope = (closed_norm - open_norm) / (closed_mm - open_mm)
      value_norm = (value_mm - closed_mm) * slope + closed_norm

      value_gripper = value_norm * 255 / 100

      if (value_gripper > 255):
          value_gripper_limited = 255
      elif (value_gripper < 0):
          value_gripper_limited = 0
      else:
          value_gripper_limited = round_value(value_gripper)
      end

      return value_gripper_limited
  end

  def round_value(value):
      value_mod = value % 1

      if(value_mod < 0.5):
          return floor(value)
      else:
          return ceil(value)
      end
  end

  def round_value_2_dec(value):
      value_x_100 = value * 100
      value_x_100_rounded = round_value(value_x_100)
      return value_x_100_rounded / 100
  end

  def clear_socket_buffer(gripper_socket="1", read_timeout = 0.1):
      rq_comm_clear_socket_buffer_enabled[rq_socket_to_index(gripper_socket)] = True
  end

  def rq_gripper_id_to_ascii(gripper_id):
      if(gripper_id == "1"):
          return 57
      elif(gripper_id == "2"):
          return 50
      elif(gripper_id == "3"):
          return 51
      elif(gripper_id == "4"):
          return 52
      end
  end

  def scale(value, rawRange, scaledRange):
      def computeSlope(inputRange, outputRange):
          outputRangeDelta = outputRange[1] - outputRange[0]
          inputRangeDelta = inputRange[1] - inputRange[0]

          if (inputRangeDelta == 0):
              return 0
          else:
              return outputRangeDelta / inputRangeDelta
          end
      end

      def computeIntercept(slope, inputRange, outputRange):
          return outputRange[0] - (slope * inputRange[0])
      end

      def clipScaledValue(outputScaledValue, outputRange):
          if (outputRange[0] < outputRange[1]):
              return clipWhenLowerLimitIsLessThanHigher(outputScaledValue, outputRange)
          else:
              return clipWhenLowerLimitIsGreaterThanHigherLimit(outputScaledValue, outputRange)
          end
      end

      def clipWhenLowerLimitIsGreaterThanHigherLimit(outputScaledValue, outputRange):
          if (outputScaledValue < outputRange[1]):
              return outputRange[1]
          elif (outputScaledValue > outputRange[0]):
              return outputRange[0]
          else:
              return outputScaledValue
          end
      end

      def clipWhenLowerLimitIsLessThanHigher(outputScaledValue, outputRange):
          if (outputScaledValue < outputRange[0]):
              return outputRange[0]
          elif (outputScaledValue > outputRange[1]):
              return outputRange[1]
          else:
              return outputScaledValue
          end
      end

      slope = computeSlope(rawRange, scaledRange)
      intercept = computeIntercept(slope, rawRange, scaledRange)
      scaledValue = slope * value + intercept
      return clipScaledValue(scaledValue, scaledRange)
  end

  def limit(value, range):
      return scale(value, range, range)
  end


  rq_init_comm_if_connected(9, "1")
  rq_init_comm_if_connected(2, "2")
  rq_init_comm_if_connected(3, "3")
  rq_init_comm_if_connected(4, "4")
  rq_print_connected_grippers()
  rq_gripper_communication_thread = run rq_gripper_communication()
  set_closed_norm(100.0, 1)
  set_open_norm(0.0, 1)
  set_closed_mm(0.0, 1)
  set_open_mm(50.0, 1)
  set_closed_norm(100.0, 2)
  set_open_norm(0.0, 2)
  set_closed_mm(0.0, 2)
  set_open_mm(50.0, 2)
  set_closed_norm(100.0, 3)
  set_open_norm(0.0, 3)
  set_closed_mm(0.0, 3)
  set_open_mm(50.0, 3)
  set_closed_norm(100.0, 4)
  set_open_norm(0.0, 4)
  set_closed_mm(0.0, 4)
  set_open_mm(50.0, 4)
  rq_current_limit_enabled = False
  while(not rq_gripper_communication_thread_started):
      sync()
  end
  # end: URCap Installation Node
  $ 1 "BeforeStart"
  $ 2 "s_open≔socket_open('192.168.0.10',30000)"
  global s_open=socket_open("192.168.0.10",30000)
  $ 3 "MoveJ"
  $ 4 "pick_pos" "breakAfter"
  movej(get_inverse_kin(p[.419428775081, -.156466791448, .391085213928, 2.180490679377, -2.261344124399, .002804421611], qnear=[0.001867666606264251, -1.1152618567100614, -2.0303900877579535, -1.5673182646379207, 1.5616202354452682, 0.045734424142303]), a=1.3962634015954636, v=1.0471975511965976)
  $ 5 "Loop s_open ≟  False "
  while (s_open  ==    False  ):
    $ 6 "s_open≔socket_open('192.168.0.10',30000)"
    global s_open=socket_open("192.168.0.10",30000)
  end
  $ 7 "robot_start≔'robot start'"
  global robot_start="robot start"
  $ 8 "server_start≔'server start'"
  global server_start="server start"
  $ 9 "part_found≔'part found'"
  global part_found="part found"
  $ 10 "part_n_found≔'part not found'"
  global part_n_found="part not found"
  $ 11 "go_ocr≔'go ocr'"
  global go_ocr="go ocr"
  $ 12 "ocr_position≔'ocr position'"
  global ocr_position="ocr position"
  $ 13 "part_placed≔'part placed'"
  global part_placed="part placed"
  $ 14 "go_pick≔'go pick'"
  global go_pick="go pick"
  $ 15 "var_2≔'0'"
  global var_2="0"
  while (True):
    $ 16 "Robot Program"
    $ 17 "toserver≔robot_start"
    global toserver=robot_start
    $ 18 "socket_send_string(toserver)"
    socket_send_string(toserver)
    $ 19 "Wait: 0.01"
    sleep(0.01)
    $ 20 "fromserver≔socket_read_string()"
    global fromserver=socket_read_string()
    $ 21 "Loop fromserver ≠ server_start"
    while (fromserver  !=  server_start):
      $ 22 "fromserver≔socket_read_string()"
      global fromserver=socket_read_string()
      $ 23 "Wait: 0.01"
      sleep(0.01)
    end
    $ 24 "campos_1"
    $ 25 "Loop"
    while (True):
      $ 26 "MoveJ"
      $ 27 "pick_pos" "breakAfter"
      movej(get_inverse_kin(p[.419428775081, -.156466791448, .391085213928, 2.180490679377, -2.261344124399, .002804421611], qnear=[0.001867666606264251, -1.1152618567100614, -2.0303900877579535, -1.5673182646379207, 1.5616202354452682, 0.045734424142303]), a=1.3962634015954636, v=1.0471975511965976, r=0.1)
      # begin: URCap Program Node
      #   Source: Robotiq_Wrist_Camera, 1.10.3.5692, Robotiq Inc.
      #   Type: Cam Locate
      $ 28 "Cam Locate"

      ###########################################
      #######VisionLocate node start########

      f=[0,0.0,0.0,0.0,0.0,0.0,0.0,0]
      object_location=p[0.0,0.0,0.0,0.0,0.0,0.0]
      feature_pose_to_restore_45951 = pp_n_1
      movej([1.1058803796768188, -1.1670668760882776, -1.9255879561053675, -1.3659794966327112, 1.0898480415344238, 1.0605189800262451])
      # Offset in translation only.
      snapshot_position_offset[3] = 0
      snapshot_position_offset[4] = 0
      snapshot_position_offset[5] = 0
      T_camera_in_flange = p[0, 0, 0, 0, 0, 0] # enlever une fois que l'enseignement du modele sera fait en faisant un movetool avec la pose de la camera dans le repere de la flange. Pour l'instant, on suppose que la camera est situee directement sur la flange.
      tool_45951 = get_T_in_base_from_flange(T_camera_in_flange)
      tool_45951 = pose_sub(tool_45951, snapshot_position_offset)
      snapshot_position = p[0.3857, 0.326079, 0.667286, -1.91141, 1.92966, -0.520215]
      textmsg("expected snapshot position : ", snapshot_position)
      diff = pose_sub(tool_45951, snapshot_position)
      textmsg("diff = ", diff)
      is_at_snapshot_position = norm([diff[0], diff[1], diff[2]]) < 0.002
      is_at_snapshot_position = is_at_snapshot_position and (norm([diff[3], diff[4], diff[5]]) < 0.005)
      textmsg("is_at_snapshot_position = ", is_at_snapshot_position)
      is_snapshot_position_offset = norm(snapshot_position_offset) != 0
      is_at_snapshot_position = is_at_snapshot_position or ignore_snapshot_position
      if not(is_at_snapshot_position):
        popup("Robot is not at Snapshot Position. Add Move instruction to Snapshot Position before Camera Locate node.. Error code: [UCC-8]", warning = False, error = True)
        halt
      end
      f_45951 = xmlrpc_server.findmodel("contextName-45951", tool_45951[0], tool_45951[1], tool_45951[2], tool_45951[3], tool_45951[4], tool_45951[5])
      cam_locate_monitor.setFindModelResult("45951", f_45951)
      canSaveImage = True
      logging_service.publish("FIND_MODEL", f_45951)
      cam_locate_monitor.setCurrentObjectIndex("45951", 0)
      # begin: URCap Program Node
      #   Source: Robotiq_Wrist_Camera, 1.10.3.5692, Robotiq Inc.
      #   Type: Cam Locate Loop
      $ 29 "For object(s) found" "noBreak"
      object_teaching_location_45951 = p[0.3972655139194614, 0.39008004971495547, 0.03268649806528501, -3.1393198709274563, 0.034253799767581854, -2.215684751352942E-5]
      feature_teaching_location_45951 = p[0.3972655139194614, 0.39008004971495547, 0.03268649806528501, -3.1394826802205165, 0.0123293219801983, -4.502308288505037E-5]
      while (not cam_locate_monitor.isCaptureNeeded("45951")):
        poseAsArray = cam_locate_monitor.getCurrentObjectPoseAsArray("45951")
        current_object_location_45951 = p[poseAsArray[0], poseAsArray[1], poseAsArray[2], poseAsArray[3], poseAsArray[4], poseAsArray[5]]
        object_location = current_object_location_45951
        f[0] = cam_locate_monitor.getNumberOfObjectsFound("45951")
        f[1] = object_location[0]
        f[2] = object_location[1]
        f[3] = object_location[2]
        f[4] = object_location[3]
        f[5] = object_location[4]
        f[6] = object_location[5]
        f[7] = cam_locate_monitor.getCurrentObjectDetectionScore("45951")
        textmsg("current_object_location = ", current_object_location_45951)
        if (norm(snapshot_position_offset) != 0):
          current_object_location_45951 = pose_add(current_object_location_45951, snapshot_position_offset)
          textmsg("current_object_location after snapshot position offset = ", current_object_location_45951)
        end
        pp_n_1 = pose_trans(current_object_location_45951, pose_trans(pose_inv(object_teaching_location_45951), feature_teaching_location_45951))
        $ 30 "lp_br≔ False " "noBreak"
        global lp_br=  False
        $ 31 "socket_send_string(part_found)" "noBreak"
        socket_send_string(part_found)
        $ 32 "target≔object_location" "noBreak"
        global target=object_location
        $ 33 "target[2] = target[2] + 0.02" "noBreak"
        target[2] = target[2] + 0.02
        $ 34 "MoveL" "noBreak"
        $ 35 "target" "noBreak"
        movel(pose_trans(p[0.0,0.0,0.0,0.0,0.0,0.0], target), a=1.2, v=0.25)
        # begin: URCap Program Node
        #   Source: Robotiq_Copilot, 1.14.5.5896, Robotiq Inc.
        #   Type: Find Surface
        $ 36 "Find Surface" "noBreak"
        rq_ft_sensor_disconnected_check()
        rq_zero_sensor()
        sleep(0.1)
        surface_found = rq_linear_search_urcap("Z-", 10.000, 0.050, 0.500, 0)
        storevar.setvariable("rq_findSurface_41898b69-db16-4f6d-856e-2ea45cbd8eeb_exitPosition", get_actual_tcp_pose())
        $ 37 "'Add Stop conditions from the Find Surface node'" "noBreak"
        # 'Add Stop conditions from the Find Surface node'
        # end: URCap Program Node
        $ 38 "vac_test≔rq_is_vacuum_obj_detected('1')" "noBreak"
        global vac_test=rq_is_vacuum_obj_detected("1")
        # begin: URCap Program Node
        #   Source: Robotiq_Grippers, 1.8.5.6286, Robotiq Inc.
        #   Type: Vacuum
        $ 39 "Vacuum Grip  (1)           " "noBreak"
        if(not rq_is_gripper_connected("1")):
            popup("A vacuum is not connected. ID: 1", "Vacuum Error", False, True, True)
        end

        rq_vacuum_grip_raw(False, 20, 40, 30, "1")

            suction_completed = rq_wait_for_vacuum_object_suction_complete("1")
            if(not suction_completed):
                rq_set_var("GTO", 0, "1")
            end

        # end: URCap Program Node
        $ 40 "vac_test≔rq_is_vacuum_obj_detected('1')" "noBreak"
        global vac_test=rq_is_vacuum_obj_detected("1")
        $ 41 "If vac_test == False " "noBreak"
        if (vac_test ==  False  ):
          # begin: URCap Program Node
          #   Source: Robotiq_Grippers, 1.8.5.6286, Robotiq Inc.
          #   Type: Vacuum
          $ 42 "Vacuum Release  (1)           " "noBreak"
          if(not rq_is_gripper_connected("1")):
              popup("A vacuum is not connected. ID: 1", "Vacuum Error", False, True, True)
          end

          if(vacuumGripCheckThread1Running):
              stopVacuumGripCheckThread(vacuumGripCheckThread1)
              vacuumGripCheckThread1Running = False
          end

          rq_vacuum_release_raw(False, 100, 60, 30, 0.05, True, "1")

          # end: URCap Program Node
          $ 43 "break" "noBreak"
          break
        end
        # begin: URCap Program Node
        #   Source: Robotiq_Copilot, 1.14.5.5896, Robotiq Inc.
        #   Type: Find Surface
        $ 44 "Find Surface" "noBreak"
        rq_ft_sensor_disconnected_check()
        rq_zero_sensor()
        sleep(0.1)
        surface_found = rq_linear_search_urcap("Z+", 10.000, 0.050, 0.050, 0)
        storevar.setvariable("rq_findSurface_06e24699-0dcd-43a2-9ade-afee589d1248_exitPosition", get_actual_tcp_pose())
        $ 45 "'Add Stop conditions from the Find Surface node'" "noBreak"
        # 'Add Stop conditions from the Find Surface node'
        # begin: URCap Program Node
        #   Source: Robotiq_Copilot, 1.14.5.5896, Robotiq Inc.
        #   Type: If surface found
        $ 46 "If surface found" "noBreak"
        if (surface_found):
          $ 47 "'Sequence if force threshold is reached'" "noBreak"
          # 'Sequence if force threshold is reached'
          # begin: URCap Program Node
          #   Source: Robotiq_Grippers, 1.8.5.6286, Robotiq Inc.
          #   Type: Vacuum
          $ 48 "Vacuum Release  (1)           " "noBreak"
          if(not rq_is_gripper_connected("1")):
              popup("A vacuum is not connected. ID: 1", "Vacuum Error", False, True, True)
          end

          if(vacuumGripCheckThread1Running):
              stopVacuumGripCheckThread(vacuumGripCheckThread1)
              vacuumGripCheckThread1Running = False
          end

          rq_vacuum_release_raw(False, 100, 60, 30, 0.05, True, "1")

          # end: URCap Program Node
          $ 49 "lp_br≔ True " "noBreak"
          global lp_br=  True
        end
        # end: URCap Program Node
        # end: URCap Program Node
        $ 50 "If lp_br == True" "noBreak"
        if (lp_br == True):
          $ 51 "break" "noBreak"
          break
        end
        $ 52 "MoveJ" "noBreak"
        $ 53 "pick_pos" "noBreak"
        movej(get_inverse_kin(p[.419428775081, -.156466791448, .391085213928, 2.180490679377, -2.261344124399, .002804421611], qnear=[0.001867666606264251, -1.1152618567100614, -2.0303900877579535, -1.5673182646379207, 1.5616202354452682, 0.045734424142303]), a=1.3962634015954636, v=1.0471975511965976)
        $ 54 "vac_test≔rq_is_vacuum_obj_detected('1')" "noBreak"
        global vac_test=rq_is_vacuum_obj_detected("1")
        $ 55 "If vac_test == False " "noBreak"
        if (vac_test ==  False  ):
          # begin: URCap Program Node
          #   Source: Robotiq_Grippers, 1.8.5.6286, Robotiq Inc.
          #   Type: Vacuum
          $ 56 "Vacuum Release  (1)           " "noBreak"
          if(not rq_is_gripper_connected("1")):
              popup("A vacuum is not connected. ID: 1", "Vacuum Error", False, True, True)
          end

          if(vacuumGripCheckThread1Running):
              stopVacuumGripCheckThread(vacuumGripCheckThread1)
              vacuumGripCheckThread1Running = False
          end

          rq_vacuum_release_raw(False, 100, 60, 30, 0.05, True, "1")

          # end: URCap Program Node
          $ 57 "break" "noBreak"
          break
        end
        $ 58 "fromserver≔socket_read_string()" "noBreak"
        global fromserver=socket_read_string()
        $ 59 "Loop fromserver ≠ go_ocr" "noBreak"
        while (fromserver  !=  go_ocr):
          $ 60 "fromserver≔socket_read_string()" "noBreak"
          global fromserver=socket_read_string()
          $ 61 "Wait: 0.01" "noBreak"
          sleep(0.01)
        end
        $ 62 "MoveJ" "noBreak"
        $ 63 "ocr_pos" "noBreak"
        movej(get_inverse_kin(p[-.092453625101, -.730464073009, .374236297511, .102971840420, 2.129473884525, -2.138994101838], qnear=[-1.4409344832049769, -1.7518847624408167, -2.363429848347799, 0.9800668954849243, 1.478285312652588, 0.12285291403532028]), a=1.3962634015954636, v=1.0471975511965976)
        $ 64 "socket_send_string(ocr_position)" "noBreak"
        socket_send_string(ocr_position)
        $ 65 "Wait: 0.5" "noBreak"
        sleep(0.5)
        $ 66 "place_position≔socket_read_binary_integer(1)" "noBreak"
        global place_position=socket_read_binary_integer(1)
        $ 67 "Loop place_position[0] ≠ 1" "noBreak"
        while (place_position[0]  !=  1):
          $ 68 "place_position≔socket_read_binary_integer(1)" "noBreak"
          global place_position=socket_read_binary_integer(1)
        end
        $ 69 "MoveJ" "noBreak"
        $ 70 "place_pos" "noBreak"
        movej(get_inverse_kin(p[-.418268335840, .159557032128, .391133158084, -2.268102149246, -2.170953829474, -.000376235848], qnear=[-3.1470142046557825, -1.1151898542987269, -2.0303662459002894, -1.5673068205462855, 1.561488389968872, 0.045806705951690674]), a=1.3962634015954636, v=1.0471975511965976, r=0.05)
        $ 71 "If  place_position[1] == 99" "noBreak"
        if ( place_position[1] == 99):
          $ 72 "MoveJ" "noBreak"
          $ 73 "failed_pos" "noBreak"
          movej(get_inverse_kin(p[-.067194965885, .511126796664, .082089930601, 2.431080906312, -1.983264260055, -.030073923490], qnear=[-4.275227133427755, -1.4694183508502405, -2.382268730794088, -0.8468087355243128, 1.5746519565582275, 1.806339979171753]), a=1.3962634015954636, v=1.0471975511965976)
        end
        $ 74 "Script: place_part.script" "noBreak"
        if(place_position[1] == 0):
          movej(p[-0.226,0.525,0.05,2.23,2.22,0])
        elif(place_position[1] == 1):
          movej(p[-0.226,0.350,0.05075,2.23,2.22,0])
        elif(place_position[1] == 2):
          movej(p[-0.226,0.175,0.05075,2.23,2.22,0])
        elif(place_position[1] == 3):
          movej(p[-0.226,-0,0.05075,2.23,2.22,0])
        elif(var_2 == "4"):
          movej(p[-0.226,-0.175,0.05075,2.23,2.22,0])
        elif(var_2 == "5"):
          movej(p[-0.226,-0.350,0.05075,2.23,2.22,0])
        elif(var_2 == "6"):
          movej(p[-0.22575,-0.525,0.05075,2.230,2.215,0])
        elif(var_2 == "7"):
          movej(p[-0.32575,0.525,0.05075,2.230,2.215,0])
        elif(var_2 == "8"):
          movej(p[-0.32575,0.350,0.05075,2.230,2.215,0])
        elif(var_2 == "9"):
          movej(p[-0.32575,0.175,0.05075,2.230,2.215,0])
        elif(var_2 == "10"):
          movej(p[-0.32575,0,0.05075,2.230,2.215,0])
        elif(var_2 == "11"):
          movej(p[-0.32575,-0.175,0.05075,2.230,2.215,0])
        elif(var_2 == "12"):
          movej(p[-0.32575,-0.350,0.05075,2.230,2.215,0])
        elif(var_2 == "13"):
          movej(p[-0.32575,-0.525,0.05075,2.230,2.215,0])
        elif(var_2 == "14"):
          movej(p[-0.42575,0.525,0.05075,2.230,2.215,0])
        elif(var_2 == "15"):
          movej(p[-0.42575,0.350,0.05075,2.230,2.215,0])
        elif(var_2 == "16"):
          movej(p[-0.42575,0.175,0.05075,2.230,2.215,0])
        elif(var_2 == "17"):
          movej(p[-0.42575,0,0.05075,2.230,2.215,0])
        elif(var_2 == "18"):
          movej(p[-0.42575,-0.175,0.05075,2.230,2.215,0])
        elif(var_2 == "19"):
          movej(p[-0.42575,-0.350,0.05075,2.230,2.215,0])
        elif(var_2 == "20"):
          movej(p[-0.42575,-0.525,0.05075,2.230,2.215,0])
        elif(var_2 == "21"):
          movej(p[-0.52575,0.525,0.05075,2.230,2.215,0])
        elif(var_2 == "22"):
          movej(p[-0.52575,0.350,0.05075,2.230,2.215,0])
        elif(var_2 == "23"):
          movej(p[-0.52575,0.175,0.05075,2.230,2.215,0])
        elif(var_2 == "24"):
          movej(p[-0.52575,0,0.05075,2.230,2.215,0])
        elif(var_2 == "25"):
          movej(p[-0.52575,-0.175,0.05075,2.230,2.215,0])
        elif(var_2 == "26"):
          movej(p[-0.52575,-0.350,0.05075,2.230,2.215,0])
        elif(var_2 == "27"):
          movej(p[-0.52575,-0.525,0.05075,2.230,2.215,0])
        elif(var_2 == "28"):
          movej(p[-0.62575,0.525,0.05075,2.230,2.215,0])
        elif(var_2 == "29"):
          movej(p[-0.62575,0.350,0.05075,2.230,2.215,0])
        elif(var_2 == "30"):
          movej(p[-0.62575,0.175,0.05075,2.230,2.215,0])
        elif(var_2 == "31"):
          movej(p[-0.62575,0,0.05075,2.230,2.215,0])
        elif(var_2 == "32"):
          movej(p[-0.62575,-0.175,0.05075,2.230,2.215,0])
        elif(var_2 == "33"):
          movej(p[-0.62575,-0.350,0.05075,2.230,2.215,0])
        elif(var_2 == "34"):
          movej(p[-0.62575,-0.525,0.05075,2.230,2.215,0])
        elif(var_2 == "35"):
          movej(p[-0.72575,0.525,0.05075,2.230,2.215,0])
        elif(var_2 == "36"):
          movej(p[-0.72575,0.350,0.05075,2.230,2.215,0])
        elif(var_2 == "37"):
          movej(p[-0.72575,0.175,0.05075,2.230,2.215,0])
        elif(var_2 == "38"):
          movej(p[-0.72575,0,0.05075,2.230,2.215,0])
        elif(var_2 == "39"):
          movej(p[-0.72575,-0.175,0.05075,2.230,2.215,0])
        elif(var_2 == "40"):
          movej(p[-0.72575,-0.350,0.05075,2.230,2.215,0])
        elif(var_2 == "41"):
          movej(p[-0.72575,-0.525,0.05075,2.230,2.215,0])
        elif(var_2 == "42"):
          movej(p[-0.82575,0.525,0.05075,2.230,2.215,0])
        elif(var_2 == "43"):
          movej(p[-0.82575,0.350,0.05075,2.230,2.215,0])
        elif(var_2 == "44"):
          movej(p[-0.82575,0.175,0.05075,2.230,2.215,0])
        elif(var_2 == "45"):
          movej(p[-0.82575,0,0.05075,2.230,2.215,0])
        elif(var_2 == "46"):
          movej(p[-0.82575,-0.175,0.05075,2.230,2.215,0])
        elif(var_2 == "47"):
          movej(p[-0.82575,-0.350,0.05075,2.230,2.215,0])
        elif(var_2 == "48"):
          movej(p[-0.82575,-0.525,0.05075,2.230,2.215,0])
        elif(var_2 == "49"):
          movej(p[-0.92575,0.525,0.05075,2.230,2.215,0])
        elif(var_2 == "50"):
          movej(p[-0.92575,0.350,0.05075,2.230,2.215,0])
        elif(var_2 == "51"):
          movej(p[-0.92575,0.175,0.05075,2.230,2.215,0])
        elif(var_2 == "52"):
          movej(p[-0.92575,0,0.05075,2.230,2.215,0])
        elif(var_2 == "53"):
          movej(p[-0.92575,-0.175,0.05075,2.230,2.215,0])
        elif(var_2 == "54"):
          movej(p[-0.92575,-0.350,0.05075,2.230,2.215,0])
        elif(var_2 == "55"):
          movej(p[-0.92575,-0.525,0.05075,2.230,2.215,0])
        elif(var_2 == "56"):
          movej(p[-1.02575,0.525,0.05075,2.230,2.215,0])
        elif(var_2 == "57"):
          movej(p[-1.02575,0.350,0.05075,2.230,2.215,0])
        elif(var_2 == "58"):
          movej(p[-1.02575,0.175,0.05075,2.230,2.215,0])
        elif(var_2 == "59"):
          movej(p[-1.02575,0,0.05075,2.230,2.215,0])
        elif(var_2 == "60"):
          movej(p[-1.02575,-0.175,0.05075,2.230,2.215,0])
        elif(var_2 == "61"):
          movej(p[-1.02575,-0.350,0.05075,2.230,2.215,0])
        elif(var_2 == "62"):
          movej(p[-1.02575,-0.525,0.05075,2.230,2.215,0])
        end
        # begin: URCap Program Node
        #   Source: Robotiq_Grippers, 1.8.5.6286, Robotiq Inc.
        #   Type: Vacuum
        $ 75 "Vacuum Release  (1)           " "noBreak"
        if(not rq_is_gripper_connected("1")):
            popup("A vacuum is not connected. ID: 1", "Vacuum Error", False, True, True)
        end

        if(vacuumGripCheckThread1Running):
            stopVacuumGripCheckThread(vacuumGripCheckThread1)
            vacuumGripCheckThread1Running = False
        end

        rq_vacuum_release_raw(False, 100, 60, 30, 0.05, True, "1")

        # end: URCap Program Node
        $ 76 "MoveJ" "noBreak"
        $ 77 "place_pos" "noBreak"
        movej(get_inverse_kin(p[-.418268335840, .159557032128, .391133158084, -2.268102149246, -2.170953829474, -.000376235848], qnear=[-3.1470142046557825, -1.1151898542987269, -2.0303662459002894, -1.5673068205462855, 1.561488389968872, 0.045806705951690674]), a=1.3962634015954636, v=1.0471975511965976, r=0.05)
        cam_locate_monitor.incrementIndex("45951")
      end
      # end: URCap Program Node
      # begin: URCap Program Node
      #   Source: Robotiq_Wrist_Camera, 1.10.3.5692, Robotiq Inc.
      #   Type: If no object found in Camera Locate
      $ 78 "If no object found" "noBreak"
      if (not cam_locate_monitor.hasFoundObjects("45951")):
        f[0] = 0
        $ 79 "Wait: 0.5" "noBreak"
        sleep(0.5)
        $ 80 "break" "noBreak"
        break
      end
      # end: URCap Program Node
      # Restore feature pose
      pp_n_1 = feature_pose_to_restore_45951

      #######VisionLocate node end########
      ###########################################

      # end: URCap Program Node
    end
    $ 81 "Popup: End"
    popup("End", "Message", False, False, blocking=True)
  end
end
